FUNCTION blockMessage 
VAR_INPUT
	error : STRING;
	
END_VAR
VAR
	strSFCErrorStep : STRING; (* Declaration*)
END_VAR

ADSLOGSTR(msgCtrlMask := ADSLOG_MSGTYPE_ERROR OR ADSLOG_MSGTYPE_LOG,
	msgFmtStr := error,
	strArg := strSFCErrorStep);

END_FUNCTION

(* stored: Version 1.1.0.1, ProductVersion 3.1.4024.12
   POU blockMessage: Id {68346874-3d2e-4f26-bed0-402040ec1f96}, SpecialFunc None *)
